// TIA Portal V21 export
TYPE "UDT_ASSI"
   STRUCT
      StsFlag : Struct   // Appoggio Flag Stato
         ErrorPb : Bool;   // Errore Connessione Profibus
         OffsetDetect : Bool;   // Richiesta Esecuzione Offest Encoder
         SetUpData : Bool;   // Richiesta Set Up
         ByPassOverTravel : Bool;   // By Pass Sicurezza FC Overtravel
         ByPassAxisAlarm : Bool;   // By Pass Allarme Assi
         Spare2 : Bool;
         Spare1 : Bool;
         SetUpEnable : Bool;   // Abilitazione Set Up Asse
         EndTrav_NEG : Bool;   // Finecorsa Negativo
         Slow_NEG : Bool;   // Rallentamento Negativo
         EndTrav_POS : Bool;   // Finecorsa Positivo
         Slow_POS : Bool;   // Rallentamento Positivo
         AppReach : Bool;   // Quota Approching Raggiunta
         PosReach : Bool;   // Quota Raggiunta
         MinSpeed : Bool;   // Finestra Minima Velocità
         MotDirection : Bool;   // Direzione Movimento 0=Avanti / 1=Indietro
         AppInProgress : Bool;   // Avvicinamento in corso
         JOGMODE_REQ : Bool;   // Modo JOG
         AUTOMODE_REQ : Bool;   // Modo Automatico
         SAUTO_REQ : Bool;   // modo semiautomatico
         Jog_P : Bool;   // Jog +
         Jog_N : Bool;   // Jog -
         PosInProgress : Bool;
         StartPosition : Bool;   // Start Posizionamento Auto
         PosReached : Bool;   // Posizione Raggiunta
         PosResch2 : Bool;
         AxesZeroSpeed : Bool;   // Asse Fermo
         CmdHalt : Bool;   // Comando Halt Asse
         DoorEnable : Bool;   // Consenso Apertura Portelle
         AxisTestMode : Bool;   // Abilita Modo Test Asse
         Finecorsa_Tutto_Basso : Bool;   // Finecorsa_Tutto_Basso
         Finecorsa_Tutto_Alto : Bool;   // Finecorsa_Tutto_Alto
      END_STRUCT;
      XRealData : Struct   // Appoggio Visualizzazione Posizione Asse
         ActPos : DInt;   // Altezza Attuale Asta Graduata(decimo di mm)
         PrgPos : DInt;   // Posizione di Destinazione
         DistToGo : DInt;   // Distanza Dal Target
         Speed : DInt;   // Velocita' Traslazione
      END_STRUCT;
      XPrgData : Struct   // Appoggio Dati set Up Asse
         ZeroOffset : DWord;   // Appoggio Offset Encoder
         Cnt_Turn : Int;   // Numero Di Impulsi Encoder Per Giro
         StepTurn : Int;   // Spostamento per Giro
         EndTravelN : DInt;   // Finecorsa Negativo
         SlowN : DInt;   // Rallentamento Negativo
         EndTravelP : DInt;   // Finecorsa Positivo
         SlowP : DInt;   // Rallentamento Positivo
         InPosItion : Int;   // Finestra In Posizione
         InApproch : Int;   // Finestra In Approching
         DeadBand : Int;   // Zona Morta
         KApp : Int;   // Guadagno Proporzionale KVApp
         VAppMax : Int;   // Massima Velocita' Avvicinamento
         KPos : Int;   // Guadagno Proporzionale Velocita' Posizionamento
         VposMax : Int;   // Massima Velocita' Di Posizionamento
         KTim : Int;   // K Spazio di Rallentamento
         Tacc : Int;   // Tempo di Accelerazione / Decelerazione
         AxesMaxSpeed : Int;   // Massima Velocità Asse (0 - 10000)
         WindMinSpeed : Int;   // Finestra Per Minima Velocità
         MinSpeedValue : Int;   // Valore Minima Velocita'
         OldAxesPos : DInt;   // Appoggio Vecchia Posizione Asse
         RowStep : Real;   // Distanza Tra Vani
         Area2 : DInt;   // Altezza Area 2
         FwErrMinValue : Int;   // Valore Massimo Errore Inseguimento
         OvrSpeedErrValue : Int;   // Valore Massimo Overspeed
         StopErrorValue : Int;   // Stop Error
         KPFollowError : Int;   // Fattore Conversione Errore Inseguimento
         AxisMaxQuote : DInt;   // Appoggio Massima Quota Encoder
         Spare : DWord;
         Spare13101 : DWord;
      END_STRUCT;
      DataTemp : Struct   // Appoggio Dati Temporanei
         RealEncCnt : DWord;   // Lettura Reale Dell' encoder
         OldValue : Word;   // Valore Vecchio del timer stamp
         Cnt_Turn : Real;   // Appoggio Impulsi Giro In Reale
         StepTurn : Real;   // Appoggio Passi Giro In Reale
         KFactor : Real;   // Fattore Conversione Cnt Encoder Step mm
         Speed_CntMin : Real;   // Velocita' espressa in Cnt / Min
         DeltaPos : DInt;   // Delta Posizione
         KSpeedFactor : DInt;   // Correzione in funzione della massima Velocità
         SelSpeedMax : DInt;   // Massima Velocità dell' asse (Calcolata)
         PickingQuote : DInt;   // Quota Prelievo strato
         LastFollowError : DInt;
         WaitingQuote : DInt;   // Quota Attesa
         QuotaPerTraslazione : DInt;   // Quota Sollevatore Dopo Prelievo Strato
         QuotaScarico : DInt;   // Quota Scarico strato
         QuotaScarico2 : DInt;   // Zona Arresto Asimetrica Limite Superiore
         AuxRealEncoderQuote : DInt;   // Appoggio Quota Reale Encoder
         spare9 : DInt;
         LevelDetect : DInt;   // Quota Rilevamento Fotocellula
      END_STRUCT;
      RampGen : Struct   // Dati Generatore Rampa
         RampFlag : Struct   // Bit Generatore Rampa
            RmpUpReq : Bool;   // Richiesta Ramp Up
            RampDwnReq : Bool;   // Richiesta Ramp Down
            RampNeed : Bool;   // Richiesta Rampa
            RmpEnable : Bool;   // Abilitazione Rampa
            Spare : Bool;
            RampUp : Bool;   // Esegue rampa Salita
            RampDown : Bool;   // Esegue Rampa Discesa
            SlopeChange : Bool;
            Spare1 : Bool;
         END_STRUCT;
         ReqSpeed : Int;   // Valore Velocita' Richiesta 0 - 1000
         ActSpeed : Int;   // Valore Velocita' Attuale
         SlopeCnt : Int;
         RampTiming : Int;   // Valore Tempo Rampa 0 - 10.00s
         RampInc : Int;   // Valore Incremento Rampa
      END_STRUCT;
      AxesSpeed : Struct
         SpeedApp : Int;   // Velocita' Avvicinamento
         SpeedPos : Int;   // Velocita' Posizionamento
         AxesSpeed : Int;   // Velocita Totale Asse
         OverRide : Int;   // Controllo OverRide
         Override1 : Int;   // Selezione Override
         Override2 : Int;   // Selezione Override
         Volume_Attuale : Int;   // Volume Attuale (Intero)
         DrvCmd : Struct
            DrvEnable : Bool;   // Abilitazione Driver
            AutoMode : Bool;
            SAutoMode : Bool;
            ManuMode : Bool;
            EmgzStop : Bool;   // Stop Emergenza
            CmdJogP : Bool;   // Cmd Jog Positivo
            CmdJogN : Bool;   // Cmd Jog Negativo
            Slow : Bool;   // Cmd Rallentamento
            CmdStop : Bool;   // Cmd Stop Asse
            FwErrorEnable : Bool;   // Abilitazione Errore Inseguimento
            StopErrEnable : Bool;   // Abilitazione Errore Stop
            OverSpeedEnable : Bool;   // Abilitazione Errore Over Speed
            FwError : Bool;   // Errore Inseguimento
            OvrSpeedError : Bool;   // Errore Over Speed
            StopError : Bool;   // Errore Stop
            Spare : Bool;   // Errore Stop
            JogMotionReq : Bool;   // Richiesta Movimento Modo Jog
            DelayJogMotionStop : Bool;   // Ritardo Disattivazione Movimento JOG
            AxisRampEnable : Bool;   // Abilitazione Rampa
            CmdMotionFw : Bool;   // Comando Avanti
            CmdMotionBk : Bool;   // Comando Indietro
            Spare6 : Bool;   // Errore Stop
            Spare7 : Bool;   // Errore Stop
            Spare8 : Bool;   // Errore Stop
            Spare9 : Bool;   // Errore Stop
            Spare10 : Bool;   // Errore Stop
            Spare11 : Bool;   // Errore Stop
            Spare12 : Bool;   // Errore Stop
            Spare13 : Bool;   // Errore Stop
            Spare14 : Bool;   // Errore Stop
            Spare15 : Bool;   // Errore Stop
            Spare16 : Bool;   // Errore Stop
         END_STRUCT;
         DriverData : Struct   // Appoggio PW Driver
            CmdWord : Word;   // Word Comando Inverter
            CmdSpeed : Int;   // Speed Word per Inverter
            CtrlWord : Word;   // Word Controllo Stato inverter
            Spare : Word;
         END_STRUCT;
         SPare : DInt;
         SPare1 : DInt;
         SPare11 : DInt;
         SPare12 : DInt;
         SPare13 : DInt;
      END_STRUCT;
      MisRequest : Struct   // Bit Richiesta Missioni
         Req1 : Bool;   // Req_Mission_1
         Req2 : Bool;   // Req_Mission_2
         Req3 : Bool;   // Req_Mission_3
         Req4 : Bool;   // Req_Mission_4
         Req5 : Bool;   // Req_Mission_5
         Req6 : Bool;   // Req_Mission_6
         Req7 : Bool;   // Req_Mission_7
         Req8 : Bool;   // Req_Mission_8
         Req9 : Bool;   // Req_Mission_9
         Req10 : Bool;   // Req_Mission_10
         Req11 : Bool;   // Req_Mission_11
         Req12 : Bool;   // Req_Mission_12
         Req13 : Bool;   // Req_Mission_13
         Req14 : Bool;   // Req_Mission_14
         Req15 : Bool;   // Req_Mission_15
         Req16 : Bool;   // Req_Mission_16
         spare : Int;
      END_STRUCT;
      MissionFlag : Struct   // Bit Ststo Missioni
         Mis_1 : Bool;   // Mission 1
         Mis_2 : Bool;   // Mission 2
         Mis_3 : Bool;   // Mission 3
         Mis_4 : Bool;   // Mission 4
         Mis_5 : Bool;   // Mission 5
         Mis_6 : Bool;   // Mission 6
         Mis_7 : Bool;   // Mission 7
         Mis_8 : Bool;   // Mission 8
         Mis_9 : Bool;   // Mission 9
         Mis_10 : Bool;   // Mission 10
         Mis_11 : Bool;   // Mission 11
         Mis_12 : Bool;   // Mission 12
         Mis_13 : Bool;   // Mission 13
         Mis_14 : Bool;   // Mission 14
         Mis_15 : Bool;   // Mission 15
         NoMissionInProgr : Bool;   // Mission In progress
      END_STRUCT;
   END_STRUCT;
END_TYPE
